# EPICS autosave request: iocBoot/sioc-esb-xps1/xpsm.req
$(P):MOTR:ABS1.VAL
$(P):MOTR:ABS2.VAL
$(P):MOTR:ABS3.VAL
$(P):MOTR:SAVED1.VAL
$(P):MOTR:SAVED2.VAL
$(P):MOTR:SAVED3.VAL
$(P):MOTR.HLM
$(P):MOTR.LLM
$(P):MOTR.DHLM
$(P):MOTR.DLLM
$(P):MOTR.TWV
$(P):MOTR.VELO
$(P):MOTR.VMAX
$(P):MOTR.VBAS
$(P):MOTR.HVEL
$(P):MOTR.ACCL
$(P):MOTR.BVEL
$(P):MOTR.BACC
$(P):MOTR.BDST
$(P):MOTR.FRAC
$(P):MOTR.JVEL
$(P):MOTR.JAR
